TYPE ST_AllocateRobotNeedlingMoveInfo :
STRUCT
	NeedleLocation		: INT;	//針位，0~49
	Box					: UINT;	//盒位，0~3
	Clip				: INT;	//使用夾爪，0~3
	Area				: STRING; // Q : 圓帶 T :轉盤

END_STRUCT
END_TYPE

(* stored: Version 1.1.0.1, ProductVersion 3.1.4024.13
   DUT ST_AllocateRobotNeedlingMoveInfo: Id {eaeaa35c-046c-479b-ada0-9dafa6361539} *)
